FUNCTION_BLOCK AUTOMATIC_POSITION_TEST
VAR_INPUT
END_VAR
VAR_OUTPUT
END_VAR
VAR
END_VAR

END_FUNCTION_BLOCK

(* stored: Version 1.1.0.1, ProductVersion 3.1.4022.18
   POU AUTOMATIC_POSITION_TEST: Id {c11d3553-987e-4a91-9492-85330ea33e6e}, SpecialFunc None *)
